// TIA Portal V18 export
// export: Created 2026-06-22T15:41:34.5521993Z, ExportSetting WithDefaults, DisplayName Totally Integrated Automation Portal, DisplayVersion V18, DisplayName TIA Portal Openness, DisplayVersion V18, DisplayName TIA Portal Version Control Interface, DisplayVersion V18, DisplayName STEP 7 Professional, DisplayVersion V18, DisplayName STEP 7 Safety, DisplayVersion V18, DisplayName WinCC Professional, DisplayVersion V18
DATA_BLOCK "DB3_Encoder"   // DB5
TITLE = Encoder HSC Data Block
{ S7_Optimized_Access := 'FALSE' }
VERSION : 0.1
// Khối dữ liệu chứa tham số và trạng thái Encoder HSC1
// stored: AutoNumber true, IsOnlyStoredInLoadMemory false, IsWriteProtectedInAS false
   VAR
      Encoder_Count_Current : DInt;
      Encoder_Count_Last : DInt;
      Encoder_Count_Delta : DInt;
      Encoder_Count_Delta_Real : Real;
      Encoder_PPR : Real := 1000.0;
      Encoder_Effective_PPR : Real;
      Encoder_SampleTime_s : Real := 0.1;
      Encoder_RPM : Real;
      Encoder_Hz_Raw : Real;
      Encoder_Hz : Real;
      Encoder_Feedback_Selected : Real;
      Encoder_Use_Feedback : Bool := true;
      Encoder_Fault : Bool;
      Encoder_Use_Fourfold : Bool := true;
      Encoder_Motor_Pole_Pairs : Real := 2.0;
      Encoder_Fallback_Active : Bool;
      Encoder_NoPulse_Count : Real;
      Encoder_NoPulse_Limit : Real := 30.0;
   END_VAR
BEGIN
END_DATA_BLOCK
